// TIA Portal project "Project2" (V17)

(* hardware
DEVICE "S7-1500/ET200MP station_1"  S7-1500 station
   slot 0: "Rail_0"  Rack  6ES7 590-1***0-0AA0
   slot 1: "PLC_1"  CPU 1516-3 PN/DP  6ES7 516-3AN01-0AB0  V2.9
      slot 3: "CPU display_1"  6ES7591-1BA00-0AA0
      slot 32768: "PROFINET interface_1"  X1
      slot 33024: "PROFINET interface_2"  X2
      slot 33280: "DP interface_1"  X3
      slot 34817: "Virtual CP interface port_1"  Virtual CP interface port  Virtual CP interface port
   slot 2: "DI 32x24VDC HF_1"  DI 32x24VDC HF  6ES7 521-1BL00-0AB0  V2.1
   slot 3: "DQ 32x24VDC/0.5A HF_1"  DQ 32x24VDC/0.5A HF  6ES7 522-1BL01-0AB0  V1.0
   slot 4: "AI 8xU/I/RTD/TC ST_1"  AI 8xU/I/RTD/TC ST  6ES7 531-7KF00-0AB0  V2.0
   slot 5: "AQ 4xU/I ST_1"  AQ 4xU/I ST  6ES7 532-5HD00-0AB0  V2.0
*)

// ===== PLC "PLC_1"  CPU 1516-3 PN/DP =====

VAR_GLOBAL   // PLC tag table "Default tag table"
   "Clock_Byte" AT %MB10 : Byte;
   "Clock_10Hz" AT %M10.0 : Bool;
   "Clock_5Hz" AT %M10.1 : Bool;
   "Clock_2.5Hz" AT %M10.2 : Bool;
   "Clock_2Hz" AT %M10.3 : Bool;
   "Clock_1.25Hz" AT %M10.4 : Bool;
   "Clock_1Hz" AT %M10.5 : Bool;
   "Clock_0.625Hz" AT %M10.6 : Bool;
   "Clock_0.5Hz" AT %M10.7 : Bool;
END_VAR

VAR_GLOBAL   // PLC tag table "saidasFisicas"
   "sinAzul" AT %Q0.1 : Bool;
END_VAR

VAR_GLOBAL   // PLC tag table "entradasFisicas"
   "bt_trava" AT %I0.1 : Bool;
END_VAR

DATA_BLOCK "SIEMENS_TESTE"   // DB1
{ S7_Optimized_Access := 'TRUE' }
VERSION : 0.1
   VAR
      booleana : Bool;
      pulsoScan0 : Bool;
      pulsoScan1 : Bool;
      inteira : Int;
      real0 : Real;
      real1 : Real;
      palavra : String;
      vetor : Array[0..9] of Int;
   END_VAR
BEGIN
END_DATA_BLOCK

// folder: System blocks/Program resources

DATA_BLOCK "c1"   // DB2
{ S7_Optimized_Access := 'TRUE' }
AUTHOR : Simatic
FAMILY : IEC
NAME : CNTR
VERSION : 1.0
// stored: InstanceOfName IEC_COUNTER
"IEC_COUNTER"
BEGIN
END_DATA_BLOCK

// folder: (top level)

FUNCTION "TESTE_VARIAVEIS_SIEMENS_LADDER" : Void   // FC1, LAD
{ S7_Optimized_Access := 'TRUE' }
VERSION : 0.1
   VAR_TEMP   // added for the SCL form of the ladder/FBD networks
      _w1 : Bool;
   END_VAR
BEGIN

REGION Network 1
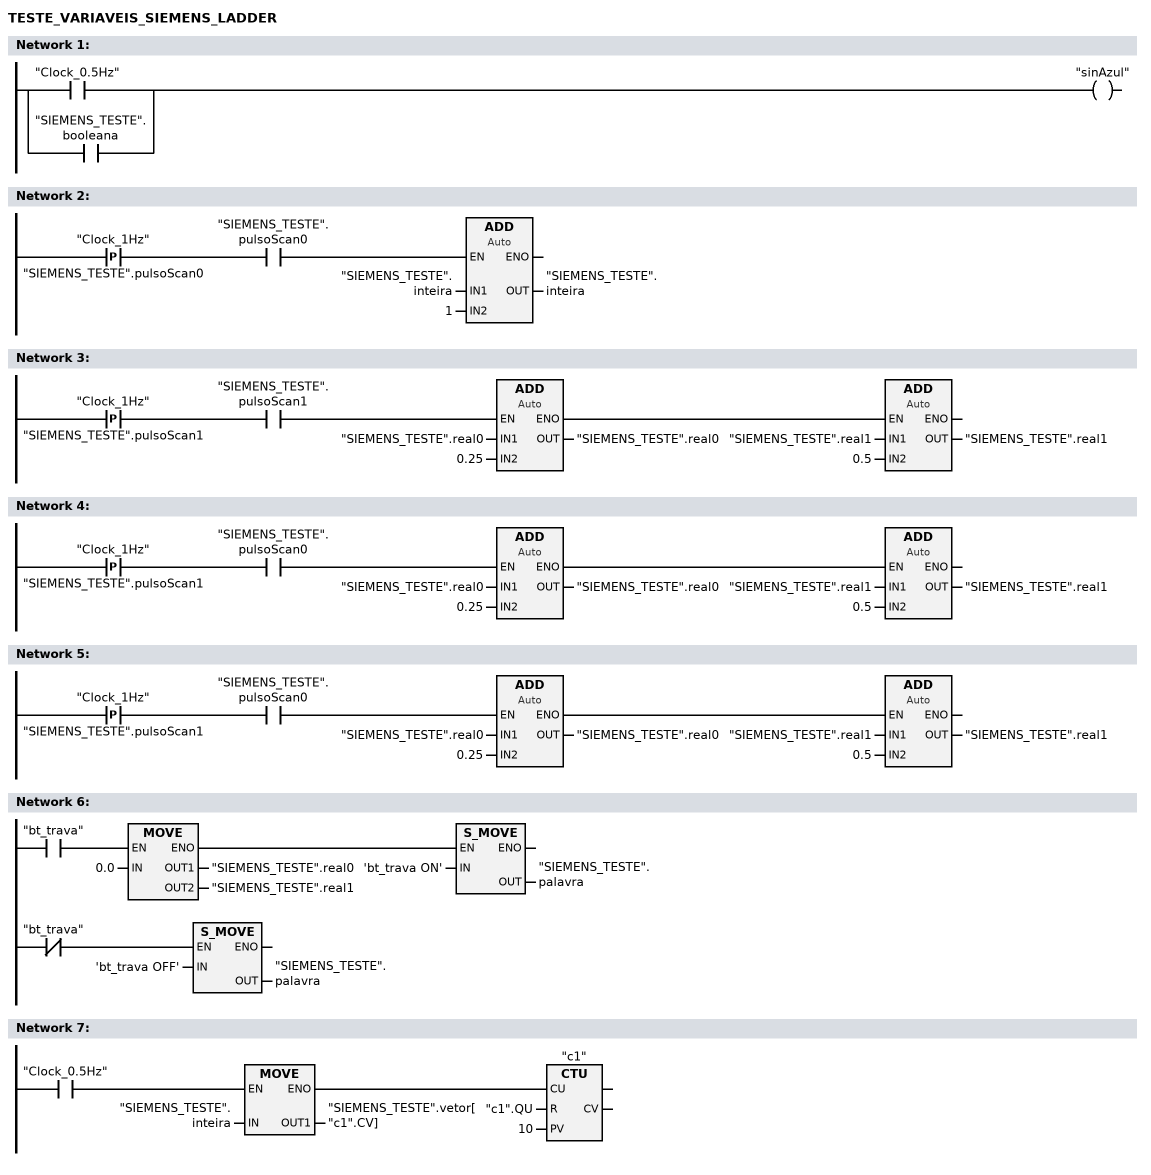
   RUNG wire#powerrail
      Contact( "Clock_0.5Hz" )
      wire#w1
      Coil( "sinAzul" )
   END_RUNG
   RUNG wire#powerrail
      Contact( "SIEMENS_TESTE".booleana )
   END_RUNG wire#w1
   // the same network as SCL:
   "sinAzul" := "Clock_0.5Hz" OR "SIEMENS_TESTE".booleana;
END_REGION

REGION Network 2
   RUNG wire#powerrail
      P_Contact(operand := "Clock_1Hz", bit := "SIEMENS_TESTE".pulsoScan0)
      Contact( "SIEMENS_TESTE".pulsoScan0 )
      Add(in1 := "SIEMENS_TESTE".inteira, in2 := 1, out => "SIEMENS_TESTE".inteira)
   END_RUNG
   // the same network as SCL:
   #_w1 := "Clock_1Hz" AND NOT "SIEMENS_TESTE".pulsoScan0;   // rising edge of "Clock_1Hz"
   "SIEMENS_TESTE".pulsoScan0 := "Clock_1Hz";
   IF #_w1 AND "SIEMENS_TESTE".pulsoScan0 THEN
       "SIEMENS_TESTE".inteira := "SIEMENS_TESTE".inteira + 1;
   END_IF;
END_REGION

REGION Network 3
   RUNG wire#powerrail
      P_Contact(operand := "Clock_1Hz", bit := "SIEMENS_TESTE".pulsoScan1)
      Contact( "SIEMENS_TESTE".pulsoScan1 )
      Add(in1 := "SIEMENS_TESTE".real0, in2 := 0.25, out => "SIEMENS_TESTE".real0)
      Add(in1 := "SIEMENS_TESTE".real1, in2 := 0.5, out => "SIEMENS_TESTE".real1)
   END_RUNG
   // the same network as SCL:
   #_w1 := "Clock_1Hz" AND NOT "SIEMENS_TESTE".pulsoScan1;   // rising edge of "Clock_1Hz"
   "SIEMENS_TESTE".pulsoScan1 := "Clock_1Hz";
   IF #_w1 AND "SIEMENS_TESTE".pulsoScan1 THEN
       "SIEMENS_TESTE".real0 := "SIEMENS_TESTE".real0 + 0.25;
       "SIEMENS_TESTE".real1 := "SIEMENS_TESTE".real1 + 0.5;
   END_IF;
END_REGION

REGION Network 4
   RUNG wire#powerrail
      P_Contact(operand := "Clock_1Hz", bit := "SIEMENS_TESTE".pulsoScan1)
      Contact( "SIEMENS_TESTE".pulsoScan0 )
      Add(in1 := "SIEMENS_TESTE".real0, in2 := 0.25, out => "SIEMENS_TESTE".real0)
      Add(in1 := "SIEMENS_TESTE".real1, in2 := 0.5, out => "SIEMENS_TESTE".real1)
   END_RUNG
   // the same network as SCL:
   #_w1 := "Clock_1Hz" AND NOT "SIEMENS_TESTE".pulsoScan1;   // rising edge of "Clock_1Hz"
   "SIEMENS_TESTE".pulsoScan1 := "Clock_1Hz";
   IF #_w1 AND "SIEMENS_TESTE".pulsoScan0 THEN
       "SIEMENS_TESTE".real0 := "SIEMENS_TESTE".real0 + 0.25;
       "SIEMENS_TESTE".real1 := "SIEMENS_TESTE".real1 + 0.5;
   END_IF;
END_REGION

REGION Network 5
   RUNG wire#powerrail
      P_Contact(operand := "Clock_1Hz", bit := "SIEMENS_TESTE".pulsoScan1)
      Contact( "SIEMENS_TESTE".pulsoScan0 )
      Add(in1 := "SIEMENS_TESTE".real0, in2 := 0.25, out => "SIEMENS_TESTE".real0)
      Add(in1 := "SIEMENS_TESTE".real1, in2 := 0.5, out => "SIEMENS_TESTE".real1)
   END_RUNG
   // the same network as SCL:
   #_w1 := "Clock_1Hz" AND NOT "SIEMENS_TESTE".pulsoScan1;   // rising edge of "Clock_1Hz"
   "SIEMENS_TESTE".pulsoScan1 := "Clock_1Hz";
   IF #_w1 AND "SIEMENS_TESTE".pulsoScan0 THEN
       "SIEMENS_TESTE".real0 := "SIEMENS_TESTE".real0 + 0.25;
       "SIEMENS_TESTE".real1 := "SIEMENS_TESTE".real1 + 0.5;
   END_IF;
END_REGION

REGION Network 6
   RUNG wire#powerrail
      Contact( "bt_trava" )
      Move(in := 0.0, out1 => "SIEMENS_TESTE".real0, out2 => "SIEMENS_TESTE".real1)
      S_Move(in := 'bt_trava ON', out => "SIEMENS_TESTE".palavra)
   END_RUNG
   RUNG wire#powerrail
      I_Contact( "bt_trava" )
      S_Move(in := 'bt_trava OFF', out => "SIEMENS_TESTE".palavra)
   END_RUNG
   // the same network as SCL:
   IF "bt_trava" THEN
       "SIEMENS_TESTE".real0 := 0.0;
       "SIEMENS_TESTE".real1 := 0.0;
       "SIEMENS_TESTE".palavra := 'bt_trava ON';
   END_IF;
   IF NOT "bt_trava" THEN "SIEMENS_TESTE".palavra := 'bt_trava OFF'; END_IF;
END_REGION

REGION Network 7
   IF "Clock_0.5Hz" THEN "SIEMENS_TESTE".vetor["c1".CV] := "SIEMENS_TESTE".inteira; END_IF;
   "c1".CTU(CU := "Clock_0.5Hz", R := "c1".QU, PV := 10);
END_REGION
END_FUNCTION

ORGANIZATION_BLOCK "Main"   // OB1, LAD, ProgramCycle
TITLE = "Main Program Sweep (Cycle)"
{ S7_Optimized_Access := 'TRUE' }
VERSION : 0.1
   VAR_INPUT
      Initial_Call : Bool;   // Initial call of this OB
      Remanence : Bool;   // =True, if remanent data are available
   END_VAR
BEGIN

REGION Network 1
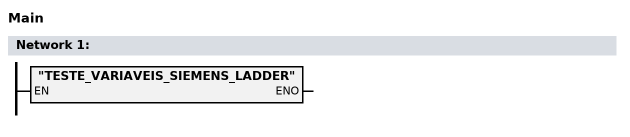
   RUNG wire#powerrail
      "TESTE_VARIAVEIS_SIEMENS_LADDER"()
   END_RUNG
   // the same network as SCL:
   "TESTE_VARIAVEIS_SIEMENS_LADDER"();
END_REGION
END_ORGANIZATION_BLOCK